{attribute 'qualified_only'}
{attribute 'strict'}
TYPE Compressor :
(
	on := 0,
	off := 1
);
END_TYPE

(* stored: Version 1.1.0.1, ProductVersion 3.1.4022.12
   DUT Compressor: Id {1dbcd13b-129b-4362-bd1e-fb515040f5f1} *)
